PROGRAM Axis05_Interlock_ST
VAR
    Always_ON      : BOOL := TRUE;
    Always_OFF     : BOOL := FALSE;
    Axis02_Safe    : BOOL;
    InRange_Home   : BOOL;
    InRange_Wait   : BOOL;
    InRange_Target : BOOL;
    InRange_Work   : BOOL;
END_VAR

VAR CONSTANT
    AXIS02_SAFE_LIMIT : REAL := 55.0;
    R_MIN             : REAL := -10.0;
    R_MAX             : REAL := 10.0;
END_VAR

// ===== 공통 조건 =====
Axis02_Safe := GVL_Axis02.Real_Position <= AXIS02_SAFE_LIMIT;

InRange_Home   := (GVL_Axis05.Home_Position_Data >= R_MIN) AND (GVL_Axis05.Home_Position_Data <= R_MAX);
InRange_Wait   := (GVL_Axis05.Wait_Position_Data >= R_MIN) AND (GVL_Axis05.Wait_Position_Data <= R_MAX);
InRange_Target := (GVL_Axis05.Target_Position_Data >= R_MIN) AND (GVL_Axis05.Target_Position_Data <= R_MAX);
InRange_Work   := (GVL_Axis05.Work_End_Position_Data >= R_MIN) AND (GVL_Axis05.Work_End_Position_Data <= R_MAX);

// ===== 개별 인터락 =====
GVL_Axis05.Home_Pos_Interlock     := Axis02_Safe OR InRange_Home;
GVL_Axis05.Wait_Pos_Interlock     := Axis02_Safe OR InRange_Wait;
GVL_Axis05.Target_Pos_Interlock   := Axis02_Safe OR InRange_Target;
GVL_Axis05.Work_End_Pos_Interlock := Axis02_Safe OR InRange_Work;
GVL_Axis05.Home_ORG_Interlock     := Axis02_Safe;

// ===== 최종 인터락 =====
GVL_Axis05.Interlock := GVL_Axis05.Home_Pos_Interlock AND 
                        GVL_Axis05.Wait_Pos_Interlock AND 
                        GVL_Axis05.Target_Pos_Interlock AND
                        GVL_Axis05.Work_End_Pos_Interlock;

END_PROGRAM

(* stored: Version 1.1.0.1, ProductVersion 3.1.4024.15
   POU Axis05_Interlock_ST: Id {d5c1cfae-6575-417a-aa96-5f28f18af423}, SpecialFunc None *)
